// TIA Portal V15 export
// export: Created 2018-12-10T18:36:37.9898147Z, ExportSetting WithDefaults, WithReadOnly, DisplayName Totally Integrated Automation Portal, DisplayVersion V15 Update 2, DisplayName TIA Portal Openness, DisplayVersion V15 Update 2, DisplayName STEP 7 Professional, DisplayVersion V15 Update 2, DisplayName STEP 7 Safety, DisplayVersion V15, DisplayName WinCC Professional, DisplayVersion V15 Update 2, DisplayName SIMATIC Visualization Architect, DisplayVersion V15 Update 1
DATA_BLOCK "FGDB_VALVENAME"   // DB89
TITLE = Geostation valve VALVENR / Geostation Ventil VALVENR
{ S7_Optimized_Access := 'FALSE' }
AUTHOR : integra
FAMILY : GF
VERSION : 0.6
// stored: AutoNumber true, CodeModifiedDate 2018-01-29T16:41:43.4527173Z, CompileDate 2018-02-20T10:24:45.6894081Z, CreationDate 2016-12-16T08:19:31.4555497Z, DBAccessibleFromOPCUA true, InstanceOfName iFG_VALVE_2D2P, InstanceOfNumber 1091, InstanceOfType FB, InterfaceModifiedDate 2018-01-24T12:18:33.5726875Z, IsConsistent true, IsKnowHowProtected false, ModifiedDate 2018-01-29T16:41:43.4527173Z, ParameterModified 2016-10-21T14:24:02.3043327Z, StructureModified 2016-10-21T14:33:02.1432809Z, UDAEnableTagReadback false
"iFG_VALVE_2D2P"
   // VAR_INPUT
   //    activateDelayTimePairMon : Bool;
   //    activateGroupMessPairMon : Bool;
   //    activateDelayTimeNoPosition : Bool;
   //    activateGroupMessNoPosition : Bool;
   //    activateStartEnableSignalsStoring : Bool;
   //    safetyStop : Bool;
   //    enableOutForward : Bool;
   //    enableOutBackward : Bool;
   //    autoForward : Bool;
   //    autoBackward : Bool;
   //    setupForward : Bool;
   //    setupBackward : Bool;
   //    usedPositionPair : Int;
   //    position_1_endForward : Bool;
   //    position_1_endBackward : Bool;
   //    position_2_endForward : Bool;
   //    position_2_endBackward : Bool;
   //    position_3_endForward : Bool;
   //    position_3_endBackward : Bool;
   //    position_4_endForward : Bool;
   //    position_4_endBackward : Bool;
   //    position_5_endForward : Bool;
   //    position_5_endBackward : Bool;
   //    position_6_endForward : Bool;
   //    position_6_endBackward : Bool;
   //    position_7_endForward : Bool;
   //    position_7_endBackward : Bool;
   //    position_8_endForward : Bool;
   //    position_8_endBackward : Bool;
   //    position_9_endForward : Bool;
   //    position_9_endBackward : Bool;
   //    position_10_endForward : Bool;
   //    position_10_endBackward : Bool;
   //    position_11_endForward : Bool;
   //    position_11_endBackward : Bool;
   //    position_12_endForward : Bool;
   //    position_12_endBackward : Bool;
   //    position_13_endForward : Bool;
   //    position_13_endBackward : Bool;
   //    position_14_endForward : Bool;
   //    position_14_endBackward : Bool;
   //    position_15_endForward : Bool;
   //    position_15_endBackward : Bool;
   //    position_16_endForward : Bool;
   //    position_16_endBackward : Bool;
   // END_VAR
   // VAR_OUTPUT
   //    qmForward : Bool;
   //    qmBackward : Bool;
   //    fault : Bool;
   //    faultExt : Bool;
   // END_VAR
   // VAR RETAIN
   //    idx : Int;
   //    sectionNumber : Int;
   //    deskNumber : Int;
   //    stationNumber : Int;
   //    dbNumber : Int;
   //    function : Int;
   //    numberInternalMessages : Int;
   //    numberExternalMessages : Int;
   //    F : Struct
   //       invalidUsedPositionPair : Bool;
   //       monitoringTimeQmForward : Bool;
   //       monitoringTimeQmBackward : Bool;
   //       groupPairMonitoring : Bool;
   //       pairMonitoring_1 : Bool;
   //       pairMonitoring_2 : Bool;
   //       pairMonitoring_3 : Bool;
   //       pairMonitoring_4 : Bool;
   //       pairMonitoring_5 : Bool;
   //       pairMonitoring_6 : Bool;
   //       pairMonitoring_7 : Bool;
   //       pairMonitoring_8 : Bool;
   //       pairMonitoring_9 : Bool;
   //       pairMonitoring_10 : Bool;
   //       pairMonitoring_11 : Bool;
   //       pairMonitoring_12 : Bool;
   //       pairMonitoring_13 : Bool;
   //       pairMonitoring_14 : Bool;
   //       pairMonitoring_15 : Bool;
   //       pairMonitoring_16 : Bool;
   //       groupNoPosition : Bool;
   //       noPostion_1 : Bool;
   //       noPostion_2 : Bool;
   //       noPostion_3 : Bool;
   //       noPostion_4 : Bool;
   //       noPostion_5 : Bool;
   //       noPostion_6 : Bool;
   //       noPostion_7 : Bool;
   //       noPostion_8 : Bool;
   //       noPostion_9 : Bool;
   //       noPostion_10 : Bool;
   //       noPostion_11 : Bool;
   //       noPostion_12 : Bool;
   //       noPostion_13 : Bool;
   //       noPostion_14 : Bool;
   //       noPostion_15 : Bool;
   //       noPostion_16 : Bool;
   //    END_STRUCT;
   //    Masks : Struct
   //       disableFault_1_8 : Byte;
   //       disableFault_9_16 : Byte;
   //       disableFault_17_24 : Byte;
   //       disableFault_25_32 : Byte;
   //       disableFault_33_40 : Byte;
   //       prodRelevantFault_1_8 : Byte;
   //       prodRelevantFault_9_16 : Byte;
   //       prodRelevantFault_17_24 : Byte;
   //       prodRelevantFault_25_32 : Byte;
   //       prodRelevantFault_33_40 : Byte;
   //    END_STRUCT;
   //    LastState : Struct
   //       fault_1_8 : Byte;
   //       fault_9_16 : Byte;
   //       fault_17_24 : Byte;
   //       fault_25_32 : Byte;
   //       fault_33_40 : Byte;
   //    END_STRUCT;
   //    IfcFGExternal : "iUDT_IFC_SYS_EXTERNAL_ALARM";
   //    Tmr : Struct
   //       s_1 { ExternalAccessible := 'False'; ExternalVisible := 'False'; ExternalWritable := 'False'; S7_SetPoint := 'True'} : Int;
   //       a_1 { ExternalAccessible := 'False'; ExternalVisible := 'False'; ExternalWritable := 'False'} : Int;
   //       s_2 { S7_SetPoint := 'True'} : Int;
   //       a_2 : Int;
   //       s_3 { S7_SetPoint := 'True'} : Int;
   //       a_3 : Int;
   //       s_4 { S7_SetPoint := 'True'} : Int;
   //       a_4 : Int;
   //       s_5 { S7_SetPoint := 'True'} : Int;
   //       a_5 : Int;
   //    END_STRUCT;
   //    ExtP : Struct
   //       setup : Bool;
   //       auto : Bool;
   //       enableIn : Bool;
   //       ack : Bool;
   //    END_STRUCT;
   //    StM : Struct
   //       fault : Bool;
   //       setup : Bool;
   //       auto : Bool;
   //       warning : Bool;
   //       eStop : Bool;
   //       safetyStop : Bool;
   //       enableIn : Bool;
   //       enableOutForward : Bool;
   //       enableOutBackward : Bool;
   //       faultPr : Bool;
   //       pairMon : Bool;
   //       specialMode : Bool;
   //       posMon : Bool;
   //       "14" : Bool;
   //       "15" : Bool;
   //       "16" : Bool;
   //       "17" : Bool;
   //       "18" : Bool;
   //       "19" : Bool;
   //       "20" : Bool;
   //       "21" : Bool;
   //       "22" : Bool;
   //       "23" : Bool;
   //       "24" : Bool;
   //       "25" : Bool;
   //       "26" : Bool;
   //       "27" : Bool;
   //       "28" : Bool;
   //       "29" : Bool;
   //       "30" : Bool;
   //       "31" : Bool;
   //       "32" : Bool;
   //    END_STRUCT;
   //    VB : Struct
   //       executabilityForward : Bool;
   //       executabilityBackward : Bool;
   //       positionEndForward : Bool;
   //       positionEndBackward : Bool;
   //       qmForward : Bool;
   //       qmBackward : Bool;
   //       "7" : Bool;
   //       "8" : Bool;
   //       "9" : Bool;
   //       "10" : Bool;
   //       "11" : Bool;
   //       "12" : Bool;
   //       "13" : Bool;
   //       "14" : Bool;
   //       "15" : Bool;
   //       "16" : Bool;
   //       "17" : Bool;
   //       "18" : Bool;
   //       "19" : Bool;
   //       "20" : Bool;
   //       "21" : Bool;
   //       "22" : Bool;
   //       "23" : Bool;
   //       "24" : Bool;
   //       "25" : Bool;
   //       "26" : Bool;
   //       "27" : Bool;
   //       "28" : Bool;
   //       "29" : Bool;
   //       "30" : Bool;
   //       "31" : Bool;
   //       "32" : Bool;
   //    END_STRUCT;
   //    VCB : Struct
   //       ack : Bool;
   //       qmForward : Bool;
   //       qmBackward : Bool;
   //       memReleaseForward : Bool;
   //       memReleaseBackward : Bool;
   //    END_STRUCT;
   //    TmrB : Struct
   //       "1_Enable" : Bool;
   //       "1_Run" : Bool;
   //       "1_Done" : Bool;
   //       "2_Enable" : Bool;
   //       "2_Run" : Bool;
   //       "2_Done" : Bool;
   //       "3_Enable" : Bool;
   //       "3_Run" : Bool;
   //       "3_Done" : Bool;
   //       "4_Enable" : Bool;
   //       "4_Run" : Bool;
   //       "4_Done" : Bool;
   //       "5_Enable" : Bool;
   //       "5_Run" : Bool;
   //       "5_Done" : Bool;
   //    END_STRUCT;
   //    D : Struct
   //       visuAck : Bool;
   //       enableIn : Bool;
   //       faultPairMonitoring_1 : Bool;
   //       faultPairMonitoring_2 : Bool;
   //       faultPairMonitoring_3 : Bool;
   //       faultPairMonitoring_4 : Bool;
   //       faultPairMonitoring_5 : Bool;
   //       faultPairMonitoring_6 : Bool;
   //       faultPairMonitoring_7 : Bool;
   //       faultPairMonitoring_8 : Bool;
   //       faultPairMonitoring_9 : Bool;
   //       faultPairMonitoring_10 : Bool;
   //       faultPairMonitoring_11 : Bool;
   //       faultPairMonitoring_12 : Bool;
   //       faultPairMonitoring_13 : Bool;
   //       faultPairMonitoring_14 : Bool;
   //       faultPairMonitoring_15 : Bool;
   //       faultPairMonitoring_16 : Bool;
   //       faultNoPosition_1 : Bool;
   //       faultNoPosition_2 : Bool;
   //       faultNoPosition_3 : Bool;
   //       faultNoPosition_4 : Bool;
   //       faultNoPosition_5 : Bool;
   //       faultNoPosition_6 : Bool;
   //       faultNoPosition_7 : Bool;
   //       faultNoPosition_8 : Bool;
   //       faultNoPosition_9 : Bool;
   //       faultNoPosition_10 : Bool;
   //       faultNoPosition_11 : Bool;
   //       faultNoPosition_12 : Bool;
   //       faultNoPosition_13 : Bool;
   //       faultNoPosition_14 : Bool;
   //       faultNoPosition_15 : Bool;
   //       faultNoPosition_16 : Bool;
   //       fault : Bool;
   //       withOverRunTime : Bool;
   //       auxFaultPairMonitoring_1 : Bool;
   //       auxFaultPairMonitoring_2 : Bool;
   //       auxFaultPairMonitoring_3 : Bool;
   //       auxFaultPairMonitoring_4 : Bool;
   //       auxFaultPairMonitoring_5 : Bool;
   //       auxFaultPairMonitoring_6 : Bool;
   //       auxFaultPairMonitoring_7 : Bool;
   //       auxFaultPairMonitoring_8 : Bool;
   //       auxFaultPairMonitoring_9 : Bool;
   //       auxFaultPairMonitoring_10 : Bool;
   //       auxFaultPairMonitoring_11 : Bool;
   //       auxFaultPairMonitoring_12 : Bool;
   //       auxFaultPairMonitoring_13 : Bool;
   //       auxFaultPairMonitoring_14 : Bool;
   //       auxFaultPairMonitoring_15 : Bool;
   //       auxFaultPairMonitoring_16 : Bool;
   //       auxfaultNoPosition_1 : Bool;
   //       auxfaultNoPosition_2 : Bool;
   //       auxfaultNoPosition_3 : Bool;
   //       auxfaultNoPosition_4 : Bool;
   //       auxfaultNoPosition_5 : Bool;
   //       auxfaultNoPosition_6 : Bool;
   //       auxfaultNoPosition_7 : Bool;
   //       auxfaultNoPosition_8 : Bool;
   //       auxfaultNoPosition_9 : Bool;
   //       auxfaultNoPosition_10 : Bool;
   //       auxfaultNoPosition_11 : Bool;
   //       auxfaultNoPosition_12 : Bool;
   //       auxfaultNoPosition_13 : Bool;
   //       auxfaultNoPosition_14 : Bool;
   //       auxfaultNoPosition_15 : Bool;
   //       auxfaultNoPosition_16 : Bool;
   //       fNPosition_1_endForward : Bool;
   //       fNPosition_1_endBackward : Bool;
   //       fNPosition_2_endForward : Bool;
   //       fNPosition_2_endBackward : Bool;
   //       fNPosition_3_endForward : Bool;
   //       fNPosition_3_endBackward : Bool;
   //       fNPosition_4_endForward : Bool;
   //       fNPosition_4_endBackward : Bool;
   //       fNPosition_5_endForward : Bool;
   //       fNPosition_5_endBackward : Bool;
   //       fNPosition_6_endForward : Bool;
   //       fNPosition_6_endBackward : Bool;
   //       fNPosition_7_endForward : Bool;
   //       fNPosition_7_endBackward : Bool;
   //       fNPosition_8_endForward : Bool;
   //       fNPosition_8_endBackward : Bool;
   //       fNPosition_9_endForward : Bool;
   //       fNPosition_9_endBackward : Bool;
   //       fNPosition_10_endForward : Bool;
   //       fNPosition_10_endBackward : Bool;
   //       fNPosition_11_endForward : Bool;
   //       fNPosition_11_endBackward : Bool;
   //       fNPosition_12_endForward : Bool;
   //       fNPosition_12_endBackward : Bool;
   //       fNPosition_13_endForward : Bool;
   //       fNPosition_13_endBackward : Bool;
   //       fNPosition_14_endForward : Bool;
   //       fNPosition_14_endBackward : Bool;
   //       fNPosition_15_endForward : Bool;
   //       fNPosition_15_endBackward : Bool;
   //       fNPosition_16_endForward : Bool;
   //       fNPosition_16_endBackward : Bool;
   //    END_STRUCT;
   //    V : Struct
   //       runtime : UInt;
   //    END_STRUCT;
   // END_VAR
BEGIN
END_DATA_BLOCK
